// TIA Portal V20 export
// export: Created 2026-07-15T01:49:22.9166942Z, ExportSetting WithDefaults, DisplayName Totally Integrated Automation Portal, DisplayVersion V20 Update 5, DisplayName TIA Portal Openness, DisplayVersion V20 Update 4, DisplayName TIA Portal Version Control Interface, DisplayVersion V20 Update 5, DisplayName SINAMICS Startdrive Advanced, DisplayVersion V20, DisplayName SINAMICS DCC, DisplayVersion V20, DisplayName SINAMICS Startdrive G130, G150, S120, S150, SINAMICS MV, G220, S200, S210, DisplayVersion V20, DisplayName SINAMICS Startdrive G110M, G120, G120C, G120D, G120P, G115D, DisplayVersion V20, DisplayName STEP 7 Professional, DisplayVersion V20 Update 5, DisplayName STEP 7 Safety, DisplayVersion V20 Update 2, DisplayName WinCC Basic/Comfort/Advanced, DisplayVersion V20 Update 5, DisplayName WinCC Unified, DisplayVersion V20 Update 5
DATA_BLOCK "MotorStarterInst8"   // DB11
VERSION : 0.1
// stored: AutoNumber true, DBAccessibleFromOPCUA true, InstanceOfName MotorStarter, InstanceOfType FB
"MotorStarter"
   // VAR RETAIN
   //    IO { S7_SetPoint := 'True'} : "MotorIOSet";
   // END_VAR
   // VAR
   //    RisingEdgeFlags : Array[0..3] of Bool;
   //    NegitiveSignalEdge : Array[0..1] of Bool;
   //    HrTotaliserTimerReset : Bool;
   //    EnableUPSTimeMS : DInt;
   //    ShutdownTimeMS : DInt;
   //    FTTimeMS : DInt;
   //    FaultTripTimer { S7_SetPoint := 'True'} : TON_TIME;
   //    FTSTimer { S7_SetPoint := 'True'} : TON_TIME;
   //    EnableUpstreamTimer { S7_SetPoint := 'True'} : TON_TIME;
   //    InHandReqPreStart { S7_SetPoint := 'True'} : TON_TIME;
   //    ShutdownTimer { S7_SetPoint := 'True'} : TON_TIME;
   //    GeneralDelayTimer { S7_SetPoint := 'True'} : TON_TIME;
   // END_VAR
   // VAR RETAIN
   //    HrTotaliserTimer { S7_SetPoint := 'True'} : TONR_TIME;
   // END_VAR
   // VAR
   //    RecentStartSignal : TOF_TIME;
   //    PreStartMemory : Bool;
   //    HandNegEdge : Bool;
   //    HandPosEdge : Bool;
   // END_VAR
BEGIN
   IO.InHand := FALSE;
   IO.AutoStartSignal := FALSE;
   IO.HandStartSignal := FALSE;
   IO.RunningFB := FALSE;
   IO.FaultFB := FALSE;
   IO.SystemHealthy := TRUE;
   IO.PreStartDone := FALSE;
   IO.InhibitMotor := FALSE;
   IO.FaultReset := FALSE;
   IO.FTTime := 3.0;
   IO.EnableUPSTime := 2.0;
   IO.FaultActive := FALSE;
   IO.Run := FALSE;
   IO.UPSEnable := FALSE;
   IO.FTR := FALSE;
   IO.FTS := FALSE;
   IO.HrsRun := 12;
   IO.Telemetry := 0;
   IO.Alarm := 16#0000;
   IO."Name" := 'Overband Magnet Unit';
   IO.HandIntervention := FALSE;
   IO.RecentStart := FALSE;
   IO.TryRunMotor := FALSE;
   IO.Shutdown := FALSE;
   IO.ShutdownComplete := TRUE;
   IO.ShutdownTime := 2.0;
   IO.StopMotor := FALSE;
   HrTotaliserTimer.PT := T#1H;
   HrTotaliserTimer.IN := FALSE;
END_DATA_BLOCK
